// TIA Portal V17 export
// export: Created 2025-03-07T09:16:45.6631924Z, ExportSetting WithDefaults, DisplayName Totally Integrated Automation Portal, DisplayVersion V17 Update 8, DisplayName TIA Portal Openness, DisplayVersion V17 Update 8, DisplayName TIA Portal Version Control Interface, DisplayVersion V17, DisplayName SINAMICS Startdrive Advanced, DisplayVersion V17 SP2, DisplayName SINAMICS Startdrive G110M, G120, G120C, G120D, G120P, G115D, DisplayVersion V17 SP2, DisplayName SINAMICS Startdrive G130, G150, S120, S150, SINAMICS MV, S210, DisplayVersion V17 SP2, DisplayName STEP 7 Professional, DisplayVersion V17 Update 8, DisplayName SINUMERIK ONE STEP 7 Toolbox, DisplayVersion V17 Update 12, DisplayName SINUMERIK 840D sl STEP 7 Toolbox, DisplayVersion V17 Update 12, DisplayName STEP 7 Safety, DisplayVersion V17 Update 6, DisplayName WinCC Advanced, DisplayVersion V17 Update 8
FUNCTION "FC2800_UNIT_01_FIXTURE_4" : Void   // FC2800, LAD
TITLE = FIXTURE 1
{ S7_Optimized_Access := 'FALSE' }
AUTHOR : ETXETAR
VERSION : 1.0
// stored: AutoNumber false, IsIECCheckEnabled false, SetENOAutomatically false, UDAEnableTagReadback false
   VAR CONSTANT
      FC_NUMBER : DInt := 2800;
   END_VAR
   VAR_TEMP   // added for the SCL form of the ladder/FBD networks
      _w1 : Bool;
      _w2 : Bool;
      _w3 : Bool;
      _w4 : Bool;
      _w5 : Bool;
   END_VAR
BEGIN

REGION Network 1: PART A PRESENT INPUT
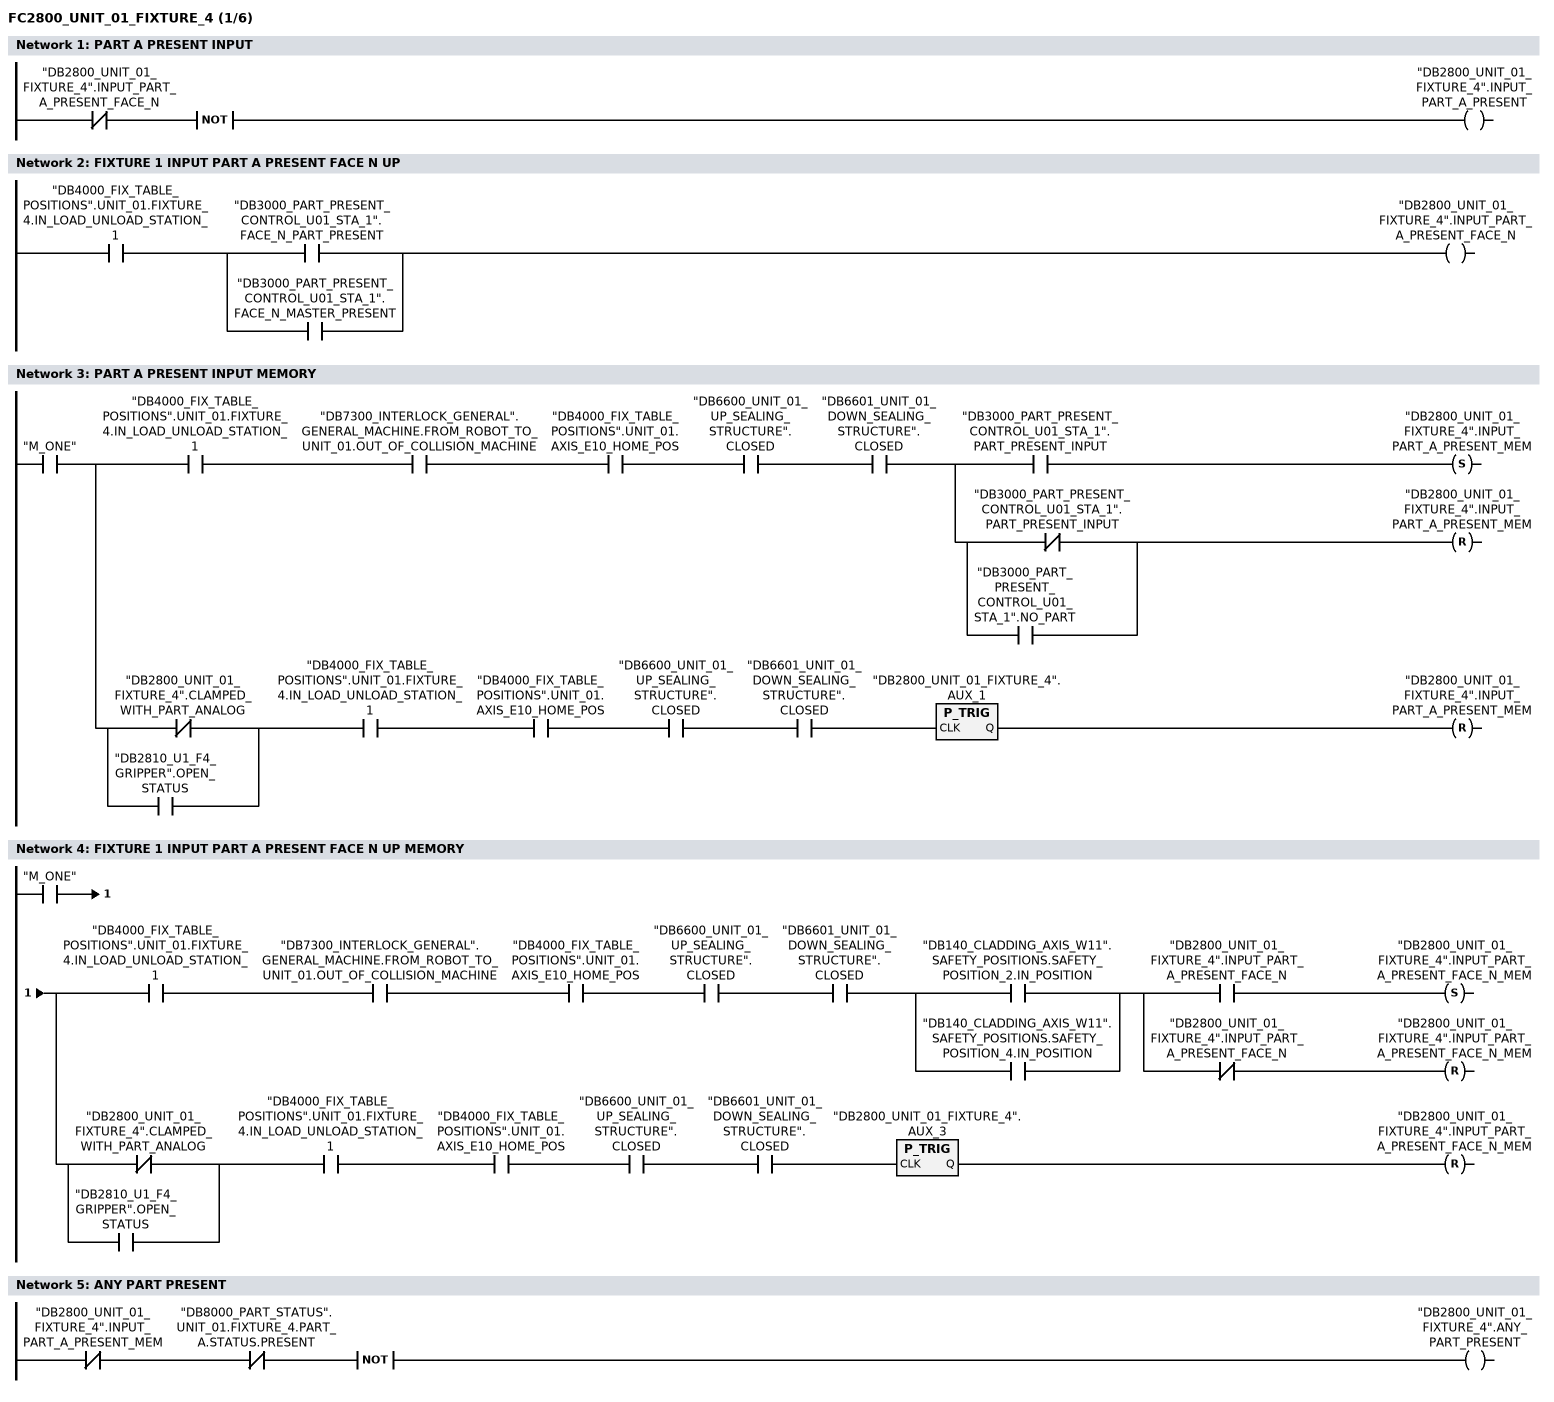
   RUNG wire#powerrail
      I_Contact( "DB2800_UNIT_01_FIXTURE_4".INPUT_PART_A_PRESENT_FACE_N )
      Not()
      Coil( "DB2800_UNIT_01_FIXTURE_4".INPUT_PART_A_PRESENT )
   END_RUNG
   // the same network as SCL:
   "DB2800_UNIT_01_FIXTURE_4".INPUT_PART_A_PRESENT := NOT (NOT "DB2800_UNIT_01_FIXTURE_4".INPUT_PART_A_PRESENT_FACE_N);
END_REGION

REGION Network 2: FIXTURE 1 INPUT PART A PRESENT FACE N UP
   RUNG wire#powerrail
      Contact( "DB4000_FIX_TABLE_POSITIONS".UNIT_01.FIXTURE_4.IN_LOAD_UNLOAD_STATION_1 )
      wire#w1
      Contact( "DB3000_PART_PRESENT_CONTROL_U01_STA_1".FACE_N_PART_PRESENT )
      wire#w2
      Coil( "DB2800_UNIT_01_FIXTURE_4".INPUT_PART_A_PRESENT_FACE_N )
   END_RUNG
   RUNG wire#w1
      Contact( "DB3000_PART_PRESENT_CONTROL_U01_STA_1".FACE_N_MASTER_PRESENT )
   END_RUNG wire#w2
   // the same network as SCL:
   "DB2800_UNIT_01_FIXTURE_4".INPUT_PART_A_PRESENT_FACE_N := "DB4000_FIX_TABLE_POSITIONS".UNIT_01.FIXTURE_4.IN_LOAD_UNLOAD_STATION_1 AND ("DB3000_PART_PRESENT_CONTROL_U01_STA_1".FACE_N_PART_PRESENT OR "DB3000_PART_PRESENT_CONTROL_U01_STA_1".FACE_N_MASTER_PRESENT);
END_REGION

REGION Network 3: PART A PRESENT INPUT MEMORY
   RUNG wire#powerrail
      Contact( "M_ONE" )
      wire#w1
      Contact( "DB4000_FIX_TABLE_POSITIONS".UNIT_01.FIXTURE_4.IN_LOAD_UNLOAD_STATION_1 )
      Contact( "DB7300_INTERLOCK_GENERAL".GENERAL_MACHINE.FROM_ROBOT_TO_UNIT_01.OUT_OF_COLLISION_MACHINE )
      Contact( "DB4000_FIX_TABLE_POSITIONS".UNIT_01.AXIS_E10_HOME_POS )
      Contact( "DB6600_UNIT_01_UP_SEALING_STRUCTURE".CLOSED )
      Contact( "DB6601_UNIT_01_DOWN_SEALING_STRUCTURE".CLOSED )
      wire#w2
      Contact( "DB3000_PART_PRESENT_CONTROL_U01_STA_1".PART_PRESENT_INPUT )
      S_Coil( "DB2800_UNIT_01_FIXTURE_4".INPUT_PART_A_PRESENT_MEM )
   END_RUNG
   RUNG wire#w2
      I_Contact( "DB3000_PART_PRESENT_CONTROL_U01_STA_1".PART_PRESENT_INPUT )
      wire#w3
      R_Coil( "DB2800_UNIT_01_FIXTURE_4".INPUT_PART_A_PRESENT_MEM )
   END_RUNG
   RUNG wire#w2
      Contact( "DB3000_PART_PRESENT_CONTROL_U01_STA_1".NO_PART )
   END_RUNG wire#w3
   RUNG wire#w1
      I_Contact( "DB2800_UNIT_01_FIXTURE_4".CLAMPED_WITH_PART_ANALOG )
      wire#w4
      Contact( "DB4000_FIX_TABLE_POSITIONS".UNIT_01.FIXTURE_4.IN_LOAD_UNLOAD_STATION_1 )
      Contact( "DB4000_FIX_TABLE_POSITIONS".UNIT_01.AXIS_E10_HOME_POS )
      Contact( "DB6600_UNIT_01_UP_SEALING_STRUCTURE".CLOSED )
      Contact( "DB6601_UNIT_01_DOWN_SEALING_STRUCTURE".CLOSED )
      P_Trig( "DB2800_UNIT_01_FIXTURE_4".AUX_1 )
      R_Coil( "DB2800_UNIT_01_FIXTURE_4".INPUT_PART_A_PRESENT_MEM )
   END_RUNG
   RUNG wire#w1
      Contact( "DB2810_U1_F4_GRIPPER".OPEN_STATUS )
   END_RUNG wire#w4
   // the same network as SCL:
   #_w1 := "M_ONE" AND "DB4000_FIX_TABLE_POSITIONS".UNIT_01.FIXTURE_4.IN_LOAD_UNLOAD_STATION_1 AND "DB7300_INTERLOCK_GENERAL".GENERAL_MACHINE.FROM_ROBOT_TO_UNIT_01.OUT_OF_COLLISION_MACHINE AND "DB4000_FIX_TABLE_POSITIONS".UNIT_01.AXIS_E10_HOME_POS AND "DB6600_UNIT_01_UP_SEALING_STRUCTURE".CLOSED AND "DB6601_UNIT_01_DOWN_SEALING_STRUCTURE".CLOSED;
   IF #_w1 AND "DB3000_PART_PRESENT_CONTROL_U01_STA_1".PART_PRESENT_INPUT THEN
       "DB2800_UNIT_01_FIXTURE_4".INPUT_PART_A_PRESENT_MEM := TRUE;
   END_IF;
   IF #_w1 AND (NOT "DB3000_PART_PRESENT_CONTROL_U01_STA_1".PART_PRESENT_INPUT OR "DB3000_PART_PRESENT_CONTROL_U01_STA_1".NO_PART) THEN
       "DB2800_UNIT_01_FIXTURE_4".INPUT_PART_A_PRESENT_MEM := FALSE;
   END_IF;
   #_w2 := "M_ONE" AND (NOT "DB2800_UNIT_01_FIXTURE_4".CLAMPED_WITH_PART_ANALOG OR "DB2810_U1_F4_GRIPPER".OPEN_STATUS) AND "DB4000_FIX_TABLE_POSITIONS".UNIT_01.FIXTURE_4.IN_LOAD_UNLOAD_STATION_1 AND "DB4000_FIX_TABLE_POSITIONS".UNIT_01.AXIS_E10_HOME_POS AND "DB6600_UNIT_01_UP_SEALING_STRUCTURE".CLOSED AND "DB6601_UNIT_01_DOWN_SEALING_STRUCTURE".CLOSED;
   #_w3 := #_w2 AND NOT "DB2800_UNIT_01_FIXTURE_4".AUX_1;   // rising edge
   "DB2800_UNIT_01_FIXTURE_4".AUX_1 := #_w2;
   IF #_w3 THEN "DB2800_UNIT_01_FIXTURE_4".INPUT_PART_A_PRESENT_MEM := FALSE; END_IF;
END_REGION

REGION Network 4: FIXTURE 1 INPUT PART A PRESENT FACE N UP MEMORY
   RUNG wire#powerrail
      Contact( "M_ONE" )
      wire#w1
      Contact( "DB4000_FIX_TABLE_POSITIONS".UNIT_01.FIXTURE_4.IN_LOAD_UNLOAD_STATION_1 )
      Contact( "DB7300_INTERLOCK_GENERAL".GENERAL_MACHINE.FROM_ROBOT_TO_UNIT_01.OUT_OF_COLLISION_MACHINE )
      Contact( "DB4000_FIX_TABLE_POSITIONS".UNIT_01.AXIS_E10_HOME_POS )
      Contact( "DB6600_UNIT_01_UP_SEALING_STRUCTURE".CLOSED )
      Contact( "DB6601_UNIT_01_DOWN_SEALING_STRUCTURE".CLOSED )
      wire#w2
      Contact( "DB140_CLADDING_AXIS_W11".SAFETY_POSITIONS.SAFETY_POSITION_2.IN_POSITION )
      wire#w3
      Contact( "DB2800_UNIT_01_FIXTURE_4".INPUT_PART_A_PRESENT_FACE_N )
      S_Coil( "DB2800_UNIT_01_FIXTURE_4".INPUT_PART_A_PRESENT_FACE_N_MEM )
   END_RUNG
   RUNG wire#w2
      Contact( "DB140_CLADDING_AXIS_W11".SAFETY_POSITIONS.SAFETY_POSITION_4.IN_POSITION )
   END_RUNG wire#w3
   RUNG wire#w3
      I_Contact( "DB2800_UNIT_01_FIXTURE_4".INPUT_PART_A_PRESENT_FACE_N )
      R_Coil( "DB2800_UNIT_01_FIXTURE_4".INPUT_PART_A_PRESENT_FACE_N_MEM )
   END_RUNG
   RUNG wire#w1
      I_Contact( "DB2800_UNIT_01_FIXTURE_4".CLAMPED_WITH_PART_ANALOG )
      wire#w4
      Contact( "DB4000_FIX_TABLE_POSITIONS".UNIT_01.FIXTURE_4.IN_LOAD_UNLOAD_STATION_1 )
      Contact( "DB4000_FIX_TABLE_POSITIONS".UNIT_01.AXIS_E10_HOME_POS )
      Contact( "DB6600_UNIT_01_UP_SEALING_STRUCTURE".CLOSED )
      Contact( "DB6601_UNIT_01_DOWN_SEALING_STRUCTURE".CLOSED )
      P_Trig( "DB2800_UNIT_01_FIXTURE_4".AUX_3 )
      R_Coil( "DB2800_UNIT_01_FIXTURE_4".INPUT_PART_A_PRESENT_FACE_N_MEM )
   END_RUNG
   RUNG wire#w1
      Contact( "DB2810_U1_F4_GRIPPER".OPEN_STATUS )
   END_RUNG wire#w4
   // the same network as SCL:
   #_w1 := "M_ONE" AND "DB4000_FIX_TABLE_POSITIONS".UNIT_01.FIXTURE_4.IN_LOAD_UNLOAD_STATION_1 AND "DB7300_INTERLOCK_GENERAL".GENERAL_MACHINE.FROM_ROBOT_TO_UNIT_01.OUT_OF_COLLISION_MACHINE AND "DB4000_FIX_TABLE_POSITIONS".UNIT_01.AXIS_E10_HOME_POS AND "DB6600_UNIT_01_UP_SEALING_STRUCTURE".CLOSED AND "DB6601_UNIT_01_DOWN_SEALING_STRUCTURE".CLOSED AND ("DB140_CLADDING_AXIS_W11".SAFETY_POSITIONS.SAFETY_POSITION_2.IN_POSITION OR "DB140_CLADDING_AXIS_W11".SAFETY_POSITIONS.SAFETY_POSITION_4.IN_POSITION);
   IF #_w1 AND "DB2800_UNIT_01_FIXTURE_4".INPUT_PART_A_PRESENT_FACE_N THEN
       "DB2800_UNIT_01_FIXTURE_4".INPUT_PART_A_PRESENT_FACE_N_MEM := TRUE;
   END_IF;
   IF #_w1 AND NOT "DB2800_UNIT_01_FIXTURE_4".INPUT_PART_A_PRESENT_FACE_N THEN
       "DB2800_UNIT_01_FIXTURE_4".INPUT_PART_A_PRESENT_FACE_N_MEM := FALSE;
   END_IF;
   #_w2 := "M_ONE" AND (NOT "DB2800_UNIT_01_FIXTURE_4".CLAMPED_WITH_PART_ANALOG OR "DB2810_U1_F4_GRIPPER".OPEN_STATUS) AND "DB4000_FIX_TABLE_POSITIONS".UNIT_01.FIXTURE_4.IN_LOAD_UNLOAD_STATION_1 AND "DB4000_FIX_TABLE_POSITIONS".UNIT_01.AXIS_E10_HOME_POS AND "DB6600_UNIT_01_UP_SEALING_STRUCTURE".CLOSED AND "DB6601_UNIT_01_DOWN_SEALING_STRUCTURE".CLOSED;
   #_w3 := #_w2 AND NOT "DB2800_UNIT_01_FIXTURE_4".AUX_3;   // rising edge
   "DB2800_UNIT_01_FIXTURE_4".AUX_3 := #_w2;
   IF #_w3 THEN "DB2800_UNIT_01_FIXTURE_4".INPUT_PART_A_PRESENT_FACE_N_MEM := FALSE; END_IF;
END_REGION

REGION Network 5: ANY PART PRESENT
   RUNG wire#powerrail
      I_Contact( "DB2800_UNIT_01_FIXTURE_4".INPUT_PART_A_PRESENT_MEM )
      I_Contact( "DB8000_PART_STATUS".UNIT_01.FIXTURE_4.PART_A.STATUS.PRESENT )
      Not()
      Coil( "DB2800_UNIT_01_FIXTURE_4".ANY_PART_PRESENT )
   END_RUNG
   // the same network as SCL:
   "DB2800_UNIT_01_FIXTURE_4".ANY_PART_PRESENT := NOT (NOT "DB2800_UNIT_01_FIXTURE_4".INPUT_PART_A_PRESENT_MEM AND NOT "DB8000_PART_STATUS".UNIT_01.FIXTURE_4.PART_A.STATUS.PRESENT);
END_REGION

REGION Network 6: CLAMPED WITH PART A
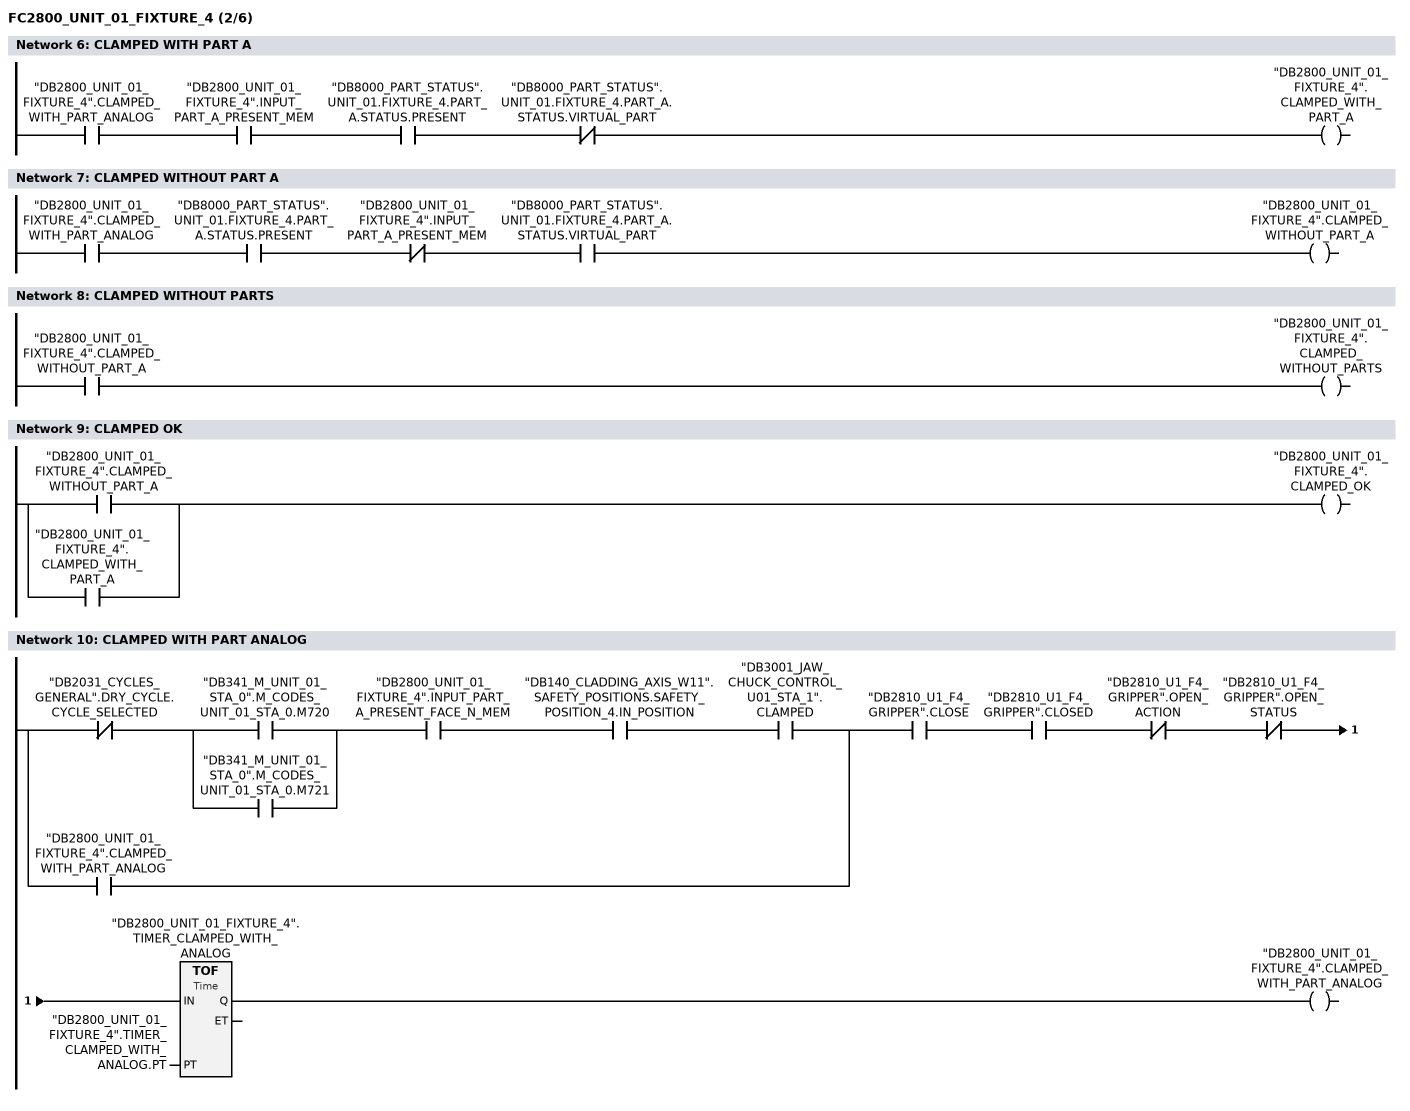
   RUNG wire#powerrail
      Contact( "DB2800_UNIT_01_FIXTURE_4".CLAMPED_WITH_PART_ANALOG )
      Contact( "DB2800_UNIT_01_FIXTURE_4".INPUT_PART_A_PRESENT_MEM )
      Contact( "DB8000_PART_STATUS".UNIT_01.FIXTURE_4.PART_A.STATUS.PRESENT )
      I_Contact( "DB8000_PART_STATUS".UNIT_01.FIXTURE_4.PART_A.STATUS.VIRTUAL_PART )
      Coil( "DB2800_UNIT_01_FIXTURE_4".CLAMPED_WITH_PART_A )
   END_RUNG
   // the same network as SCL:
   "DB2800_UNIT_01_FIXTURE_4".CLAMPED_WITH_PART_A := "DB2800_UNIT_01_FIXTURE_4".CLAMPED_WITH_PART_ANALOG AND "DB2800_UNIT_01_FIXTURE_4".INPUT_PART_A_PRESENT_MEM AND "DB8000_PART_STATUS".UNIT_01.FIXTURE_4.PART_A.STATUS.PRESENT AND NOT "DB8000_PART_STATUS".UNIT_01.FIXTURE_4.PART_A.STATUS.VIRTUAL_PART;
END_REGION

REGION Network 7: CLAMPED WITHOUT PART A
   RUNG wire#powerrail
      Contact( "DB2800_UNIT_01_FIXTURE_4".CLAMPED_WITH_PART_ANALOG )
      Contact( "DB8000_PART_STATUS".UNIT_01.FIXTURE_4.PART_A.STATUS.PRESENT )
      I_Contact( "DB2800_UNIT_01_FIXTURE_4".INPUT_PART_A_PRESENT_MEM )
      Contact( "DB8000_PART_STATUS".UNIT_01.FIXTURE_4.PART_A.STATUS.VIRTUAL_PART )
      Coil( "DB2800_UNIT_01_FIXTURE_4".CLAMPED_WITHOUT_PART_A )
   END_RUNG
   // the same network as SCL:
   "DB2800_UNIT_01_FIXTURE_4".CLAMPED_WITHOUT_PART_A := "DB2800_UNIT_01_FIXTURE_4".CLAMPED_WITH_PART_ANALOG AND "DB8000_PART_STATUS".UNIT_01.FIXTURE_4.PART_A.STATUS.PRESENT AND NOT "DB2800_UNIT_01_FIXTURE_4".INPUT_PART_A_PRESENT_MEM AND "DB8000_PART_STATUS".UNIT_01.FIXTURE_4.PART_A.STATUS.VIRTUAL_PART;
END_REGION

REGION Network 8: CLAMPED WITHOUT PARTS
   RUNG wire#powerrail
      Contact( "DB2800_UNIT_01_FIXTURE_4".CLAMPED_WITHOUT_PART_A )
      Coil( "DB2800_UNIT_01_FIXTURE_4".CLAMPED_WITHOUT_PARTS )
   END_RUNG
   // the same network as SCL:
   "DB2800_UNIT_01_FIXTURE_4".CLAMPED_WITHOUT_PARTS := "DB2800_UNIT_01_FIXTURE_4".CLAMPED_WITHOUT_PART_A;
END_REGION

REGION Network 9: CLAMPED OK
   RUNG wire#powerrail
      Contact( "DB2800_UNIT_01_FIXTURE_4".CLAMPED_WITHOUT_PART_A )
      wire#w1
      Coil( "DB2800_UNIT_01_FIXTURE_4".CLAMPED_OK )
   END_RUNG
   RUNG wire#powerrail
      Contact( "DB2800_UNIT_01_FIXTURE_4".CLAMPED_WITH_PART_A )
   END_RUNG wire#w1
   // the same network as SCL:
   "DB2800_UNIT_01_FIXTURE_4".CLAMPED_OK := "DB2800_UNIT_01_FIXTURE_4".CLAMPED_WITHOUT_PART_A OR "DB2800_UNIT_01_FIXTURE_4".CLAMPED_WITH_PART_A;
END_REGION

REGION Network 10: CLAMPED WITH PART ANALOG
   RUNG wire#powerrail
      I_Contact( "DB2031_CYCLES_GENERAL".DRY_CYCLE.CYCLE_SELECTED )
      wire#w1
      Contact( "DB341_M_UNIT_01_STA_0".M_CODES_UNIT_01_STA_0.M720 )
      wire#w2
      Contact( "DB2800_UNIT_01_FIXTURE_4".INPUT_PART_A_PRESENT_FACE_N_MEM )
      Contact( "DB140_CLADDING_AXIS_W11".SAFETY_POSITIONS.SAFETY_POSITION_4.IN_POSITION )
      Contact( "DB3001_JAW_CHUCK_CONTROL_U01_STA_1".CLAMPED )
      wire#w3
      Contact( "DB2810_U1_F4_GRIPPER".CLOSE )
      Contact( "DB2810_U1_F4_GRIPPER".CLOSED )
      I_Contact( "DB2810_U1_F4_GRIPPER".OPEN_ACTION )
      I_Contact( "DB2810_U1_F4_GRIPPER".OPEN_STATUS )
      { S7_Templates := "time_type := Time" } "DB2800_UNIT_01_FIXTURE_4".TIMER_CLAMPED_WITH_ANALOG.TOF(pt := "DB2800_UNIT_01_FIXTURE_4".TIMER_CLAMPED_WITH_ANALOG.PT, et =>)
      Coil( "DB2800_UNIT_01_FIXTURE_4".CLAMPED_WITH_PART_ANALOG )
   END_RUNG
   RUNG wire#w1
      Contact( "DB341_M_UNIT_01_STA_0".M_CODES_UNIT_01_STA_0.M721 )
   END_RUNG wire#w2
   RUNG wire#powerrail
      Contact( "DB2800_UNIT_01_FIXTURE_4".CLAMPED_WITH_PART_ANALOG )
   END_RUNG wire#w3
   // the same network as SCL:
   "DB2800_UNIT_01_FIXTURE_4".TIMER_CLAMPED_WITH_ANALOG.TOF(IN := ((NOT "DB2031_CYCLES_GENERAL".DRY_CYCLE.CYCLE_SELECTED AND ("DB341_M_UNIT_01_STA_0".M_CODES_UNIT_01_STA_0.M720 OR "DB341_M_UNIT_01_STA_0".M_CODES_UNIT_01_STA_0.M721) AND "DB2800_UNIT_01_FIXTURE_4".INPUT_PART_A_PRESENT_FACE_N_MEM AND "DB140_CLADDING_AXIS_W11".SAFETY_POSITIONS.SAFETY_POSITION_4.IN_POSITION AND "DB3001_JAW_CHUCK_CONTROL_U01_STA_1".CLAMPED) OR "DB2800_UNIT_01_FIXTURE_4".CLAMPED_WITH_PART_ANALOG) AND "DB2810_U1_F4_GRIPPER".CLOSE AND "DB2810_U1_F4_GRIPPER".CLOSED AND NOT "DB2810_U1_F4_GRIPPER".OPEN_ACTION AND NOT "DB2810_U1_F4_GRIPPER".OPEN_STATUS,
                           PT := "DB2800_UNIT_01_FIXTURE_4".TIMER_CLAMPED_WITH_ANALOG.PT);
   "DB2800_UNIT_01_FIXTURE_4".CLAMPED_WITH_PART_ANALOG := "DB2800_UNIT_01_FIXTURE_4".TIMER_CLAMPED_WITH_ANALOG.Q;
END_REGION

REGION Network 11: CLAMPED WITHOUT PART ANALOG
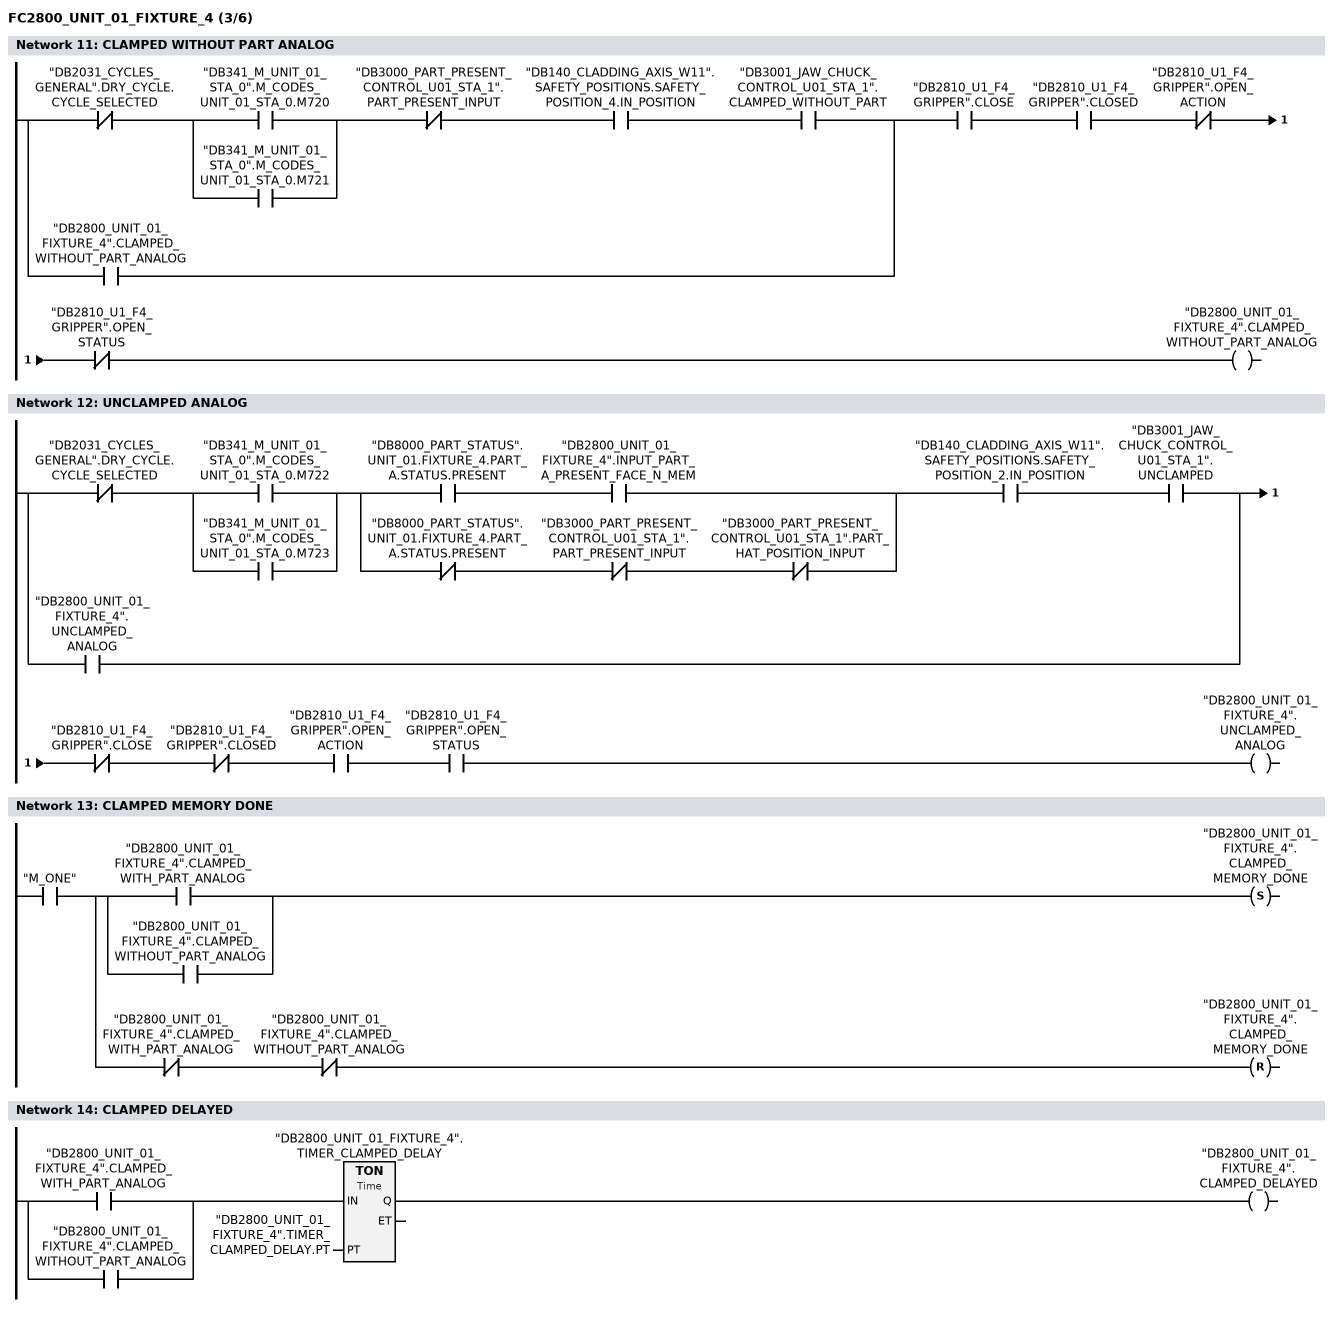
   RUNG wire#powerrail
      I_Contact( "DB2031_CYCLES_GENERAL".DRY_CYCLE.CYCLE_SELECTED )
      wire#w1
      Contact( "DB341_M_UNIT_01_STA_0".M_CODES_UNIT_01_STA_0.M720 )
      wire#w2
      I_Contact( "DB3000_PART_PRESENT_CONTROL_U01_STA_1".PART_PRESENT_INPUT )
      Contact( "DB140_CLADDING_AXIS_W11".SAFETY_POSITIONS.SAFETY_POSITION_4.IN_POSITION )
      Contact( "DB3001_JAW_CHUCK_CONTROL_U01_STA_1".CLAMPED_WITHOUT_PART )
      wire#w3
      Contact( "DB2810_U1_F4_GRIPPER".CLOSE )
      Contact( "DB2810_U1_F4_GRIPPER".CLOSED )
      I_Contact( "DB2810_U1_F4_GRIPPER".OPEN_ACTION )
      I_Contact( "DB2810_U1_F4_GRIPPER".OPEN_STATUS )
      Coil( "DB2800_UNIT_01_FIXTURE_4".CLAMPED_WITHOUT_PART_ANALOG )
   END_RUNG
   RUNG wire#w1
      Contact( "DB341_M_UNIT_01_STA_0".M_CODES_UNIT_01_STA_0.M721 )
   END_RUNG wire#w2
   RUNG wire#powerrail
      Contact( "DB2800_UNIT_01_FIXTURE_4".CLAMPED_WITHOUT_PART_ANALOG )
   END_RUNG wire#w3
   // the same network as SCL:
   "DB2800_UNIT_01_FIXTURE_4".CLAMPED_WITHOUT_PART_ANALOG := ((NOT "DB2031_CYCLES_GENERAL".DRY_CYCLE.CYCLE_SELECTED AND ("DB341_M_UNIT_01_STA_0".M_CODES_UNIT_01_STA_0.M720 OR "DB341_M_UNIT_01_STA_0".M_CODES_UNIT_01_STA_0.M721) AND NOT "DB3000_PART_PRESENT_CONTROL_U01_STA_1".PART_PRESENT_INPUT AND "DB140_CLADDING_AXIS_W11".SAFETY_POSITIONS.SAFETY_POSITION_4.IN_POSITION AND "DB3001_JAW_CHUCK_CONTROL_U01_STA_1".CLAMPED_WITHOUT_PART) OR "DB2800_UNIT_01_FIXTURE_4".CLAMPED_WITHOUT_PART_ANALOG) AND "DB2810_U1_F4_GRIPPER".CLOSE AND "DB2810_U1_F4_GRIPPER".CLOSED AND NOT "DB2810_U1_F4_GRIPPER".OPEN_ACTION AND NOT "DB2810_U1_F4_GRIPPER".OPEN_STATUS;
END_REGION

REGION Network 12: UNCLAMPED ANALOG
   RUNG wire#powerrail
      I_Contact( "DB2031_CYCLES_GENERAL".DRY_CYCLE.CYCLE_SELECTED )
      wire#w1
      Contact( "DB341_M_UNIT_01_STA_0".M_CODES_UNIT_01_STA_0.M722 )
      wire#w2
      Contact( "DB8000_PART_STATUS".UNIT_01.FIXTURE_4.PART_A.STATUS.PRESENT )
      Contact( "DB2800_UNIT_01_FIXTURE_4".INPUT_PART_A_PRESENT_FACE_N_MEM )
      wire#w3
      Contact( "DB140_CLADDING_AXIS_W11".SAFETY_POSITIONS.SAFETY_POSITION_2.IN_POSITION )
      Contact( "DB3001_JAW_CHUCK_CONTROL_U01_STA_1".UNCLAMPED )
      wire#w4
      I_Contact( "DB2810_U1_F4_GRIPPER".CLOSE )
      I_Contact( "DB2810_U1_F4_GRIPPER".CLOSED )
      Contact( "DB2810_U1_F4_GRIPPER".OPEN_ACTION )
      Contact( "DB2810_U1_F4_GRIPPER".OPEN_STATUS )
      Coil( "DB2800_UNIT_01_FIXTURE_4".UNCLAMPED_ANALOG )
   END_RUNG
   RUNG wire#w1
      Contact( "DB341_M_UNIT_01_STA_0".M_CODES_UNIT_01_STA_0.M723 )
   END_RUNG wire#w2
   RUNG wire#w2
      I_Contact( "DB8000_PART_STATUS".UNIT_01.FIXTURE_4.PART_A.STATUS.PRESENT )
      I_Contact( "DB3000_PART_PRESENT_CONTROL_U01_STA_1".PART_PRESENT_INPUT )
      I_Contact( "DB3000_PART_PRESENT_CONTROL_U01_STA_1".PART_HAT_POSITION_INPUT )
   END_RUNG wire#w3
   RUNG wire#powerrail
      Contact( "DB2800_UNIT_01_FIXTURE_4".UNCLAMPED_ANALOG )
   END_RUNG wire#w4
   // the same network as SCL:
   "DB2800_UNIT_01_FIXTURE_4".UNCLAMPED_ANALOG := ((NOT "DB2031_CYCLES_GENERAL".DRY_CYCLE.CYCLE_SELECTED AND ("DB341_M_UNIT_01_STA_0".M_CODES_UNIT_01_STA_0.M722 OR "DB341_M_UNIT_01_STA_0".M_CODES_UNIT_01_STA_0.M723) AND (("DB8000_PART_STATUS".UNIT_01.FIXTURE_4.PART_A.STATUS.PRESENT AND "DB2800_UNIT_01_FIXTURE_4".INPUT_PART_A_PRESENT_FACE_N_MEM) OR (NOT "DB8000_PART_STATUS".UNIT_01.FIXTURE_4.PART_A.STATUS.PRESENT AND NOT "DB3000_PART_PRESENT_CONTROL_U01_STA_1".PART_PRESENT_INPUT AND NOT "DB3000_PART_PRESENT_CONTROL_U01_STA_1".PART_HAT_POSITION_INPUT)) AND "DB140_CLADDING_AXIS_W11".SAFETY_POSITIONS.SAFETY_POSITION_2.IN_POSITION AND "DB3001_JAW_CHUCK_CONTROL_U01_STA_1".UNCLAMPED) OR "DB2800_UNIT_01_FIXTURE_4".UNCLAMPED_ANALOG) AND NOT "DB2810_U1_F4_GRIPPER".CLOSE AND NOT "DB2810_U1_F4_GRIPPER".CLOSED AND "DB2810_U1_F4_GRIPPER".OPEN_ACTION AND "DB2810_U1_F4_GRIPPER".OPEN_STATUS;
END_REGION

REGION Network 13: CLAMPED MEMORY DONE
   RUNG wire#powerrail
      Contact( "M_ONE" )
      wire#w1
      Contact( "DB2800_UNIT_01_FIXTURE_4".CLAMPED_WITH_PART_ANALOG )
      wire#w2
      S_Coil( "DB2800_UNIT_01_FIXTURE_4".CLAMPED_MEMORY_DONE )
   END_RUNG
   RUNG wire#w1
      Contact( "DB2800_UNIT_01_FIXTURE_4".CLAMPED_WITHOUT_PART_ANALOG )
   END_RUNG wire#w2
   RUNG wire#w1
      I_Contact( "DB2800_UNIT_01_FIXTURE_4".CLAMPED_WITH_PART_ANALOG )
      I_Contact( "DB2800_UNIT_01_FIXTURE_4".CLAMPED_WITHOUT_PART_ANALOG )
      R_Coil( "DB2800_UNIT_01_FIXTURE_4".CLAMPED_MEMORY_DONE )
   END_RUNG
   // the same network as SCL:
   IF "M_ONE" AND ("DB2800_UNIT_01_FIXTURE_4".CLAMPED_WITH_PART_ANALOG OR "DB2800_UNIT_01_FIXTURE_4".CLAMPED_WITHOUT_PART_ANALOG) THEN
       "DB2800_UNIT_01_FIXTURE_4".CLAMPED_MEMORY_DONE := TRUE;
   END_IF;
   IF "M_ONE" AND NOT "DB2800_UNIT_01_FIXTURE_4".CLAMPED_WITH_PART_ANALOG AND NOT "DB2800_UNIT_01_FIXTURE_4".CLAMPED_WITHOUT_PART_ANALOG THEN
       "DB2800_UNIT_01_FIXTURE_4".CLAMPED_MEMORY_DONE := FALSE;
   END_IF;
END_REGION

REGION Network 14: CLAMPED DELAYED
   RUNG wire#powerrail
      Contact( "DB2800_UNIT_01_FIXTURE_4".CLAMPED_WITH_PART_ANALOG )
      wire#w1
      { S7_Templates := "time_type := Time" } "DB2800_UNIT_01_FIXTURE_4".TIMER_CLAMPED_DELAY.TON(pt := "DB2800_UNIT_01_FIXTURE_4".TIMER_CLAMPED_DELAY.PT, et =>)
      Coil( "DB2800_UNIT_01_FIXTURE_4".CLAMPED_DELAYED )
   END_RUNG
   RUNG wire#powerrail
      Contact( "DB2800_UNIT_01_FIXTURE_4".CLAMPED_WITHOUT_PART_ANALOG )
   END_RUNG wire#w1
   // the same network as SCL:
   "DB2800_UNIT_01_FIXTURE_4".TIMER_CLAMPED_DELAY.TON(IN := "DB2800_UNIT_01_FIXTURE_4".CLAMPED_WITH_PART_ANALOG OR "DB2800_UNIT_01_FIXTURE_4".CLAMPED_WITHOUT_PART_ANALOG,
                           PT := "DB2800_UNIT_01_FIXTURE_4".TIMER_CLAMPED_DELAY.PT);
   "DB2800_UNIT_01_FIXTURE_4".CLAMPED_DELAYED := "DB2800_UNIT_01_FIXTURE_4".TIMER_CLAMPED_DELAY.Q;
END_REGION

REGION Network 15: ALL CNC PLC VARIABLES ZERO
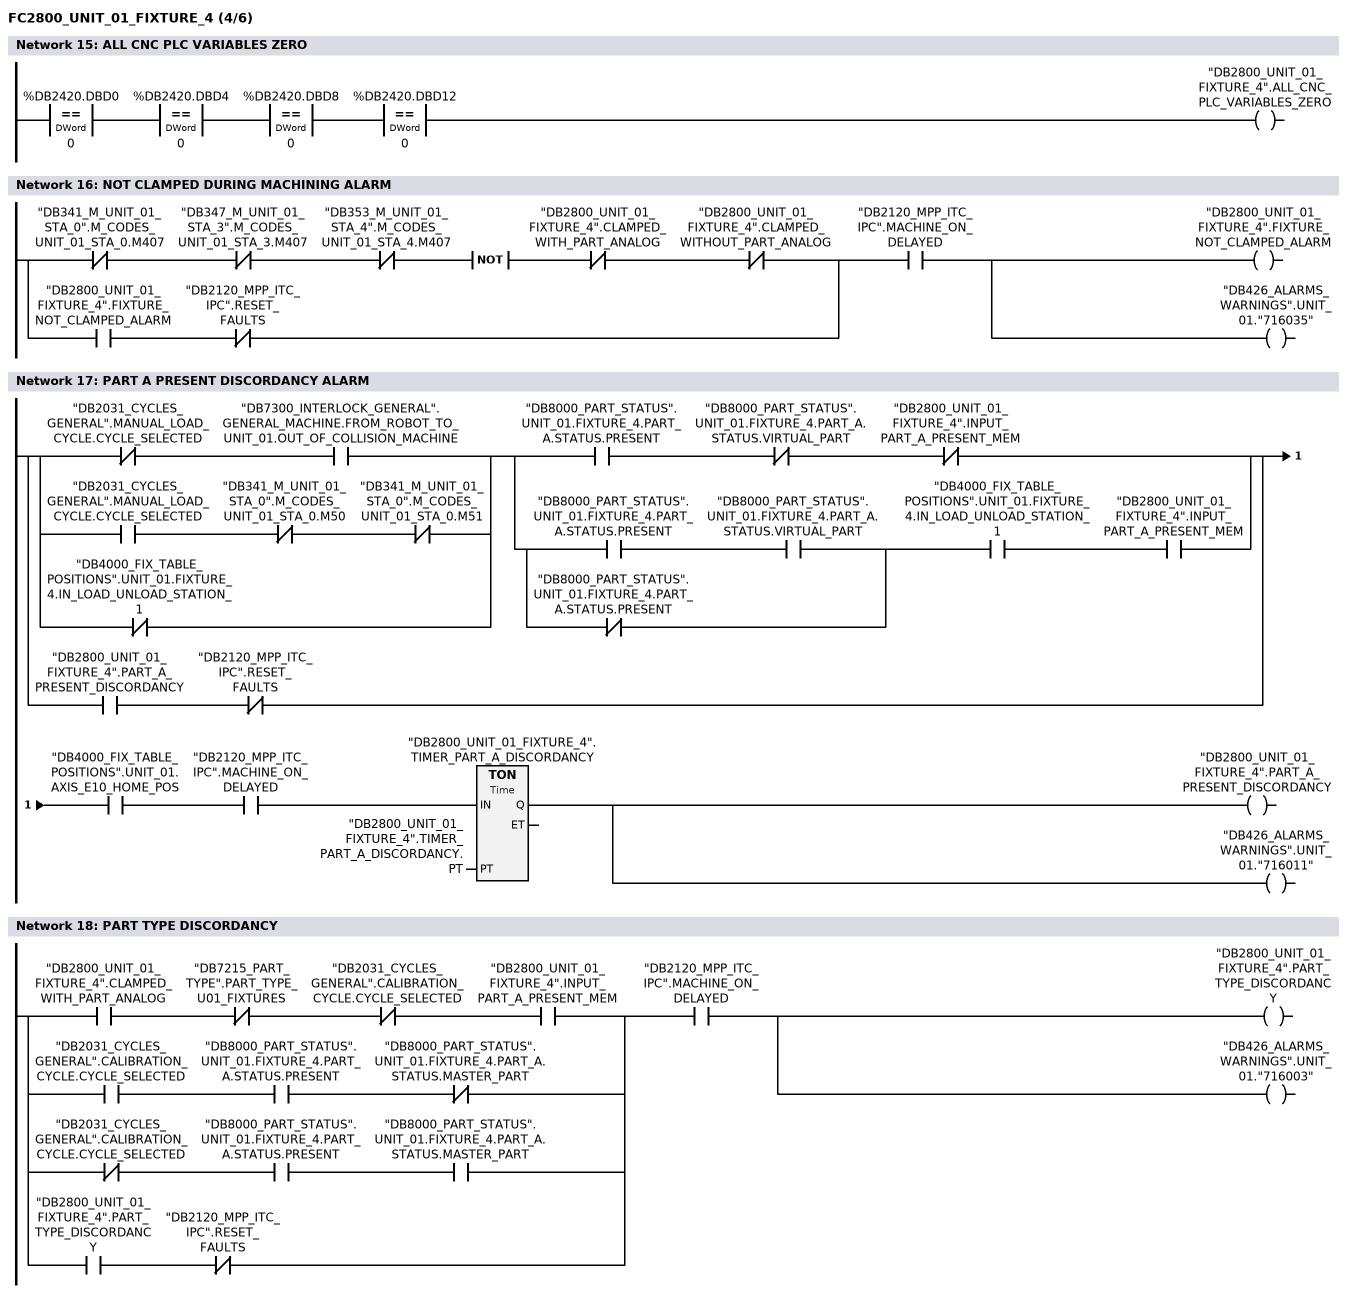
   RUNG wire#powerrail
      { S7_Templates := "SrcType := DWord" } EQ_Contact(in1 := %DB2420.DBD0, in2 := 0)
      { S7_Templates := "SrcType := DWord" } EQ_Contact(in1 := %DB2420.DBD4, in2 := 0)
      { S7_Templates := "SrcType := DWord" } EQ_Contact(in1 := %DB2420.DBD8, in2 := 0)
      { S7_Templates := "SrcType := DWord" } EQ_Contact(in1 := %DB2420.DBD12, in2 := 0)
      Coil( "DB2800_UNIT_01_FIXTURE_4".ALL_CNC_PLC_VARIABLES_ZERO )
   END_RUNG
   // the same network as SCL:
   "DB2800_UNIT_01_FIXTURE_4".ALL_CNC_PLC_VARIABLES_ZERO := (%DB2420.DBD0 = 0) AND (%DB2420.DBD4 = 0) AND (%DB2420.DBD8 = 0) AND (%DB2420.DBD12 = 0);
END_REGION

REGION Network 16: NOT CLAMPED DURING MACHINING ALARM
   RUNG wire#powerrail
      I_Contact( "DB341_M_UNIT_01_STA_0".M_CODES_UNIT_01_STA_0.M407 )
      I_Contact( "DB347_M_UNIT_01_STA_3".M_CODES_UNIT_01_STA_3.M407 )
      I_Contact( "DB353_M_UNIT_01_STA_4".M_CODES_UNIT_01_STA_4.M407 )
      Not()
      I_Contact( "DB2800_UNIT_01_FIXTURE_4".CLAMPED_WITH_PART_ANALOG )
      I_Contact( "DB2800_UNIT_01_FIXTURE_4".CLAMPED_WITHOUT_PART_ANALOG )
      wire#w1
      Contact( "DB2120_MPP_ITC_IPC".MACHINE_ON_DELAYED )
      wire#w2
      Coil( "DB2800_UNIT_01_FIXTURE_4".FIXTURE_NOT_CLAMPED_ALARM )
   END_RUNG
   RUNG wire#powerrail
      Contact( "DB2800_UNIT_01_FIXTURE_4".FIXTURE_NOT_CLAMPED_ALARM )
      I_Contact( "DB2120_MPP_ITC_IPC".RESET_FAULTS )
   END_RUNG wire#w1
   RUNG wire#w2
      Coil( "DB426_ALARMS_WARNINGS".UNIT_01."716035" )
   END_RUNG
   // the same network as SCL:
   "DB2800_UNIT_01_FIXTURE_4".FIXTURE_NOT_CLAMPED_ALARM := ((NOT (NOT "DB341_M_UNIT_01_STA_0".M_CODES_UNIT_01_STA_0.M407 AND NOT "DB347_M_UNIT_01_STA_3".M_CODES_UNIT_01_STA_3.M407 AND NOT "DB353_M_UNIT_01_STA_4".M_CODES_UNIT_01_STA_4.M407) AND NOT "DB2800_UNIT_01_FIXTURE_4".CLAMPED_WITH_PART_ANALOG AND NOT "DB2800_UNIT_01_FIXTURE_4".CLAMPED_WITHOUT_PART_ANALOG) OR ("DB2800_UNIT_01_FIXTURE_4".FIXTURE_NOT_CLAMPED_ALARM AND NOT "DB2120_MPP_ITC_IPC".RESET_FAULTS)) AND "DB2120_MPP_ITC_IPC".MACHINE_ON_DELAYED;
   "DB426_ALARMS_WARNINGS".UNIT_01."716035" := "DB2800_UNIT_01_FIXTURE_4".FIXTURE_NOT_CLAMPED_ALARM;
END_REGION

REGION Network 17: PART A PRESENT DISCORDANCY ALARM
   RUNG wire#powerrail
      I_Contact( "DB2031_CYCLES_GENERAL".MANUAL_LOAD_CYCLE.CYCLE_SELECTED )
      Contact( "DB7300_INTERLOCK_GENERAL".GENERAL_MACHINE.FROM_ROBOT_TO_UNIT_01.OUT_OF_COLLISION_MACHINE )
      wire#w1
      Contact( "DB8000_PART_STATUS".UNIT_01.FIXTURE_4.PART_A.STATUS.PRESENT )
      I_Contact( "DB8000_PART_STATUS".UNIT_01.FIXTURE_4.PART_A.STATUS.VIRTUAL_PART )
      I_Contact( "DB2800_UNIT_01_FIXTURE_4".INPUT_PART_A_PRESENT_MEM )
      wire#w2
      Contact( "DB4000_FIX_TABLE_POSITIONS".UNIT_01.AXIS_E10_HOME_POS )
      Contact( "DB2120_MPP_ITC_IPC".MACHINE_ON_DELAYED )
      { S7_Templates := "time_type := Time" } "DB2800_UNIT_01_FIXTURE_4".TIMER_PART_A_DISCORDANCY.TON(pt := "DB2800_UNIT_01_FIXTURE_4".TIMER_PART_A_DISCORDANCY.PT, et =>)
      wire#w4
      Coil( "DB2800_UNIT_01_FIXTURE_4".PART_A_PRESENT_DISCORDANCY )
   END_RUNG
   RUNG wire#powerrail
      Contact( "DB2031_CYCLES_GENERAL".MANUAL_LOAD_CYCLE.CYCLE_SELECTED )
      I_Contact( "DB341_M_UNIT_01_STA_0".M_CODES_UNIT_01_STA_0.M50 )
      I_Contact( "DB341_M_UNIT_01_STA_0".M_CODES_UNIT_01_STA_0.M51 )
   END_RUNG wire#w1
   RUNG wire#powerrail
      I_Contact( "DB4000_FIX_TABLE_POSITIONS".UNIT_01.FIXTURE_4.IN_LOAD_UNLOAD_STATION_1 )
   END_RUNG wire#w1
   RUNG wire#w1
      Contact( "DB8000_PART_STATUS".UNIT_01.FIXTURE_4.PART_A.STATUS.PRESENT )
      Contact( "DB8000_PART_STATUS".UNIT_01.FIXTURE_4.PART_A.STATUS.VIRTUAL_PART )
      wire#w3
      Contact( "DB4000_FIX_TABLE_POSITIONS".UNIT_01.FIXTURE_4.IN_LOAD_UNLOAD_STATION_1 )
      Contact( "DB2800_UNIT_01_FIXTURE_4".INPUT_PART_A_PRESENT_MEM )
   END_RUNG wire#w2
   RUNG wire#w1
      I_Contact( "DB8000_PART_STATUS".UNIT_01.FIXTURE_4.PART_A.STATUS.PRESENT )
   END_RUNG wire#w3
   RUNG wire#powerrail
      Contact( "DB2800_UNIT_01_FIXTURE_4".PART_A_PRESENT_DISCORDANCY )
      I_Contact( "DB2120_MPP_ITC_IPC".RESET_FAULTS )
   END_RUNG wire#w2
   RUNG wire#w4
      Coil( "DB426_ALARMS_WARNINGS".UNIT_01."716011" )
   END_RUNG
   // the same network as SCL:
   "DB2800_UNIT_01_FIXTURE_4".TIMER_PART_A_DISCORDANCY.TON(IN := ((((NOT "DB2031_CYCLES_GENERAL".MANUAL_LOAD_CYCLE.CYCLE_SELECTED AND "DB7300_INTERLOCK_GENERAL".GENERAL_MACHINE.FROM_ROBOT_TO_UNIT_01.OUT_OF_COLLISION_MACHINE) OR ("DB2031_CYCLES_GENERAL".MANUAL_LOAD_CYCLE.CYCLE_SELECTED AND NOT "DB341_M_UNIT_01_STA_0".M_CODES_UNIT_01_STA_0.M50 AND NOT "DB341_M_UNIT_01_STA_0".M_CODES_UNIT_01_STA_0.M51) OR NOT "DB4000_FIX_TABLE_POSITIONS".UNIT_01.FIXTURE_4.IN_LOAD_UNLOAD_STATION_1) AND (("DB8000_PART_STATUS".UNIT_01.FIXTURE_4.PART_A.STATUS.PRESENT AND NOT "DB8000_PART_STATUS".UNIT_01.FIXTURE_4.PART_A.STATUS.VIRTUAL_PART AND NOT "DB2800_UNIT_01_FIXTURE_4".INPUT_PART_A_PRESENT_MEM) OR ((("DB8000_PART_STATUS".UNIT_01.FIXTURE_4.PART_A.STATUS.PRESENT AND "DB8000_PART_STATUS".UNIT_01.FIXTURE_4.PART_A.STATUS.VIRTUAL_PART) OR NOT "DB8000_PART_STATUS".UNIT_01.FIXTURE_4.PART_A.STATUS.PRESENT) AND "DB4000_FIX_TABLE_POSITIONS".UNIT_01.FIXTURE_4.IN_LOAD_UNLOAD_STATION_1 AND "DB2800_UNIT_01_FIXTURE_4".INPUT_PART_A_PRESENT_MEM))) OR ("DB2800_UNIT_01_FIXTURE_4".PART_A_PRESENT_DISCORDANCY AND NOT "DB2120_MPP_ITC_IPC".RESET_FAULTS)) AND "DB4000_FIX_TABLE_POSITIONS".UNIT_01.AXIS_E10_HOME_POS AND "DB2120_MPP_ITC_IPC".MACHINE_ON_DELAYED,
                           PT := "DB2800_UNIT_01_FIXTURE_4".TIMER_PART_A_DISCORDANCY.PT);
   "DB2800_UNIT_01_FIXTURE_4".PART_A_PRESENT_DISCORDANCY := "DB2800_UNIT_01_FIXTURE_4".TIMER_PART_A_DISCORDANCY.Q;
   "DB426_ALARMS_WARNINGS".UNIT_01."716011" := "DB2800_UNIT_01_FIXTURE_4".TIMER_PART_A_DISCORDANCY.Q;
END_REGION

REGION Network 18: PART TYPE DISCORDANCY
   RUNG wire#powerrail
      Contact( "DB2800_UNIT_01_FIXTURE_4".CLAMPED_WITH_PART_ANALOG )
      I_Contact( "DB7215_PART_TYPE".PART_TYPE_U01_FIXTURES )
      I_Contact( "DB2031_CYCLES_GENERAL".CALIBRATION_CYCLE.CYCLE_SELECTED )
      Contact( "DB2800_UNIT_01_FIXTURE_4".INPUT_PART_A_PRESENT_MEM )
      wire#w1
      Contact( "DB2120_MPP_ITC_IPC".MACHINE_ON_DELAYED )
      wire#w2
      Coil( "DB2800_UNIT_01_FIXTURE_4".PART_TYPE_DISCORDANCY )
   END_RUNG
   RUNG wire#powerrail
      Contact( "DB2031_CYCLES_GENERAL".CALIBRATION_CYCLE.CYCLE_SELECTED )
      Contact( "DB8000_PART_STATUS".UNIT_01.FIXTURE_4.PART_A.STATUS.PRESENT )
      I_Contact( "DB8000_PART_STATUS".UNIT_01.FIXTURE_4.PART_A.STATUS.MASTER_PART )
   END_RUNG wire#w1
   RUNG wire#powerrail
      I_Contact( "DB2031_CYCLES_GENERAL".CALIBRATION_CYCLE.CYCLE_SELECTED )
      Contact( "DB8000_PART_STATUS".UNIT_01.FIXTURE_4.PART_A.STATUS.PRESENT )
      Contact( "DB8000_PART_STATUS".UNIT_01.FIXTURE_4.PART_A.STATUS.MASTER_PART )
   END_RUNG wire#w1
   RUNG wire#powerrail
      Contact( "DB2800_UNIT_01_FIXTURE_4".PART_TYPE_DISCORDANCY )
      I_Contact( "DB2120_MPP_ITC_IPC".RESET_FAULTS )
   END_RUNG wire#w1
   RUNG wire#w2
      Coil( "DB426_ALARMS_WARNINGS".UNIT_01."716003" )
   END_RUNG
   // the same network as SCL:
   "DB2800_UNIT_01_FIXTURE_4".PART_TYPE_DISCORDANCY := (("DB2800_UNIT_01_FIXTURE_4".CLAMPED_WITH_PART_ANALOG AND NOT "DB7215_PART_TYPE".PART_TYPE_U01_FIXTURES AND NOT "DB2031_CYCLES_GENERAL".CALIBRATION_CYCLE.CYCLE_SELECTED AND "DB2800_UNIT_01_FIXTURE_4".INPUT_PART_A_PRESENT_MEM) OR ("DB2031_CYCLES_GENERAL".CALIBRATION_CYCLE.CYCLE_SELECTED AND "DB8000_PART_STATUS".UNIT_01.FIXTURE_4.PART_A.STATUS.PRESENT AND NOT "DB8000_PART_STATUS".UNIT_01.FIXTURE_4.PART_A.STATUS.MASTER_PART) OR (NOT "DB2031_CYCLES_GENERAL".CALIBRATION_CYCLE.CYCLE_SELECTED AND "DB8000_PART_STATUS".UNIT_01.FIXTURE_4.PART_A.STATUS.PRESENT AND "DB8000_PART_STATUS".UNIT_01.FIXTURE_4.PART_A.STATUS.MASTER_PART) OR ("DB2800_UNIT_01_FIXTURE_4".PART_TYPE_DISCORDANCY AND NOT "DB2120_MPP_ITC_IPC".RESET_FAULTS)) AND "DB2120_MPP_ITC_IPC".MACHINE_ON_DELAYED;
   "DB426_ALARMS_WARNINGS".UNIT_01."716003" := "DB2800_UNIT_01_FIXTURE_4".PART_TYPE_DISCORDANCY;
END_REGION

REGION Network 19: PART A ORIENTATED DISCORDANCY
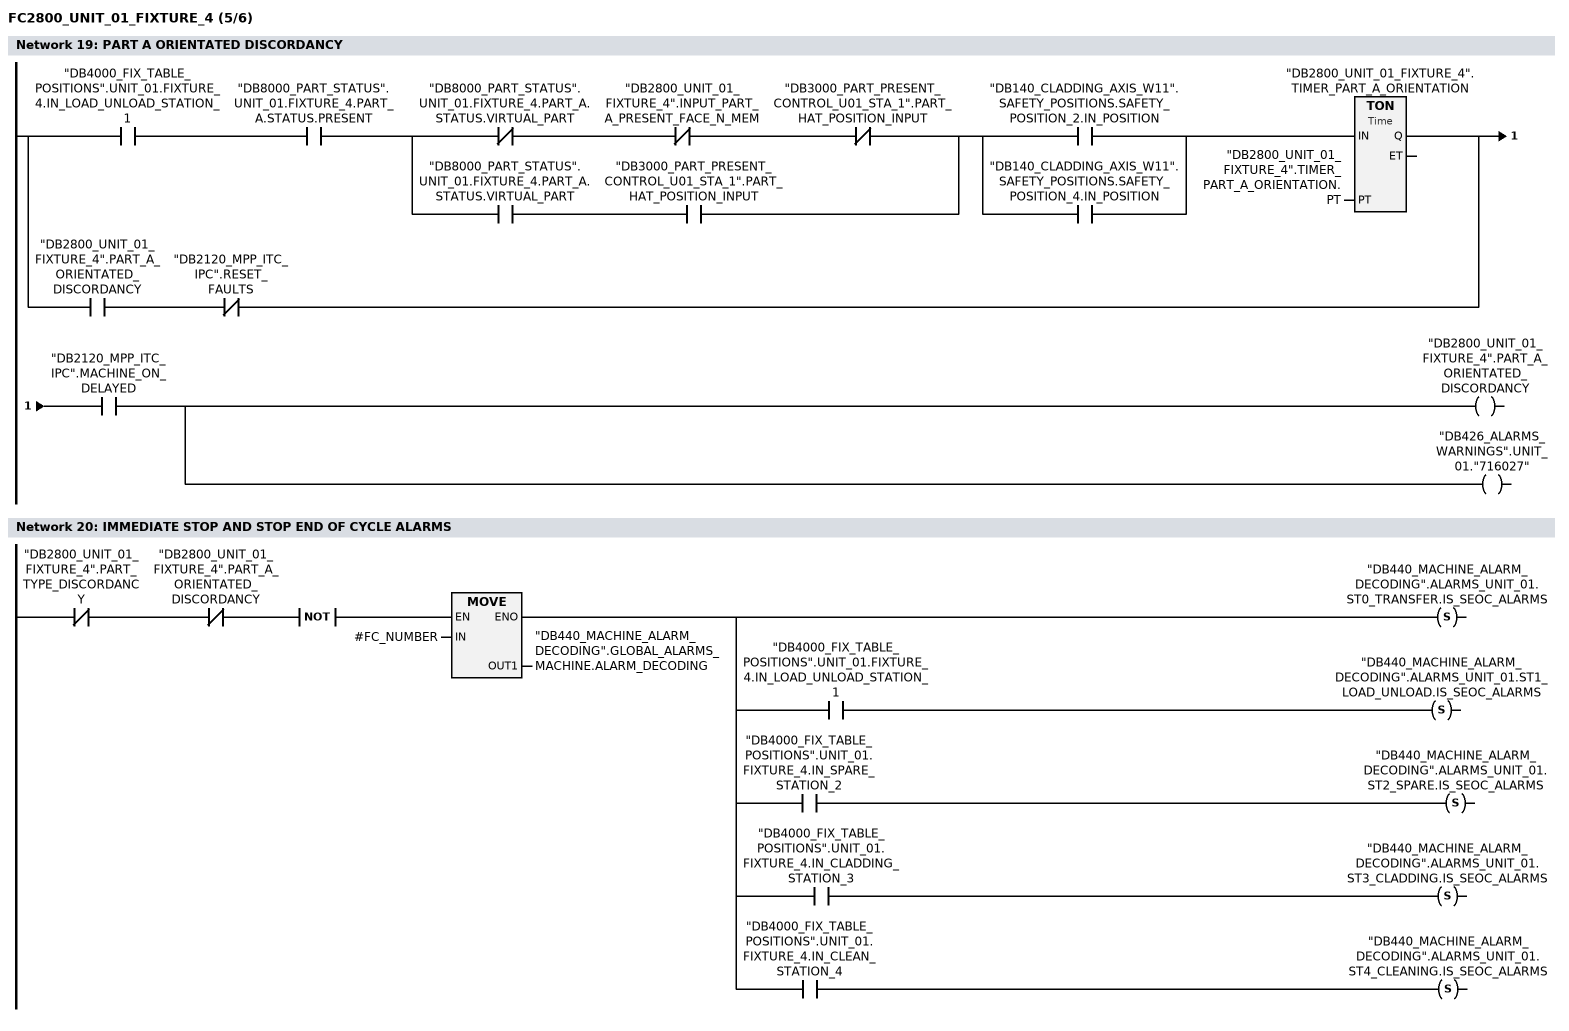
   RUNG wire#powerrail
      Contact( "DB4000_FIX_TABLE_POSITIONS".UNIT_01.FIXTURE_4.IN_LOAD_UNLOAD_STATION_1 )
      Contact( "DB8000_PART_STATUS".UNIT_01.FIXTURE_4.PART_A.STATUS.PRESENT )
      wire#w1
      I_Contact( "DB8000_PART_STATUS".UNIT_01.FIXTURE_4.PART_A.STATUS.VIRTUAL_PART )
      I_Contact( "DB2800_UNIT_01_FIXTURE_4".INPUT_PART_A_PRESENT_FACE_N_MEM )
      I_Contact( "DB3000_PART_PRESENT_CONTROL_U01_STA_1".PART_HAT_POSITION_INPUT )
      wire#w2
      Contact( "DB140_CLADDING_AXIS_W11".SAFETY_POSITIONS.SAFETY_POSITION_2.IN_POSITION )
      wire#w3
      { S7_Templates := "time_type := Time" } "DB2800_UNIT_01_FIXTURE_4".TIMER_PART_A_ORIENTATION.TON(pt := "DB2800_UNIT_01_FIXTURE_4".TIMER_PART_A_ORIENTATION.PT, et =>)
      wire#w4
      Contact( "DB2120_MPP_ITC_IPC".MACHINE_ON_DELAYED )
      wire#w5
      Coil( "DB2800_UNIT_01_FIXTURE_4".PART_A_ORIENTATED_DISCORDANCY )
   END_RUNG
   RUNG wire#w1
      Contact( "DB8000_PART_STATUS".UNIT_01.FIXTURE_4.PART_A.STATUS.VIRTUAL_PART )
      Contact( "DB3000_PART_PRESENT_CONTROL_U01_STA_1".PART_HAT_POSITION_INPUT )
   END_RUNG wire#w2
   RUNG wire#w2
      Contact( "DB140_CLADDING_AXIS_W11".SAFETY_POSITIONS.SAFETY_POSITION_4.IN_POSITION )
   END_RUNG wire#w3
   RUNG wire#powerrail
      Contact( "DB2800_UNIT_01_FIXTURE_4".PART_A_ORIENTATED_DISCORDANCY )
      I_Contact( "DB2120_MPP_ITC_IPC".RESET_FAULTS )
   END_RUNG wire#w4
   RUNG wire#w5
      Coil( "DB426_ALARMS_WARNINGS".UNIT_01."716027" )
   END_RUNG
   // the same network as SCL:
   "DB2800_UNIT_01_FIXTURE_4".TIMER_PART_A_ORIENTATION.TON(IN := "DB4000_FIX_TABLE_POSITIONS".UNIT_01.FIXTURE_4.IN_LOAD_UNLOAD_STATION_1 AND "DB8000_PART_STATUS".UNIT_01.FIXTURE_4.PART_A.STATUS.PRESENT AND ((NOT "DB8000_PART_STATUS".UNIT_01.FIXTURE_4.PART_A.STATUS.VIRTUAL_PART AND NOT "DB2800_UNIT_01_FIXTURE_4".INPUT_PART_A_PRESENT_FACE_N_MEM AND NOT "DB3000_PART_PRESENT_CONTROL_U01_STA_1".PART_HAT_POSITION_INPUT) OR ("DB8000_PART_STATUS".UNIT_01.FIXTURE_4.PART_A.STATUS.VIRTUAL_PART AND "DB3000_PART_PRESENT_CONTROL_U01_STA_1".PART_HAT_POSITION_INPUT)) AND ("DB140_CLADDING_AXIS_W11".SAFETY_POSITIONS.SAFETY_POSITION_2.IN_POSITION OR "DB140_CLADDING_AXIS_W11".SAFETY_POSITIONS.SAFETY_POSITION_4.IN_POSITION),
                           PT := "DB2800_UNIT_01_FIXTURE_4".TIMER_PART_A_ORIENTATION.PT);
   "DB2800_UNIT_01_FIXTURE_4".PART_A_ORIENTATED_DISCORDANCY := ("DB2800_UNIT_01_FIXTURE_4".TIMER_PART_A_ORIENTATION.Q OR ("DB2800_UNIT_01_FIXTURE_4".PART_A_ORIENTATED_DISCORDANCY AND NOT "DB2120_MPP_ITC_IPC".RESET_FAULTS)) AND "DB2120_MPP_ITC_IPC".MACHINE_ON_DELAYED;
   "DB426_ALARMS_WARNINGS".UNIT_01."716027" := "DB2800_UNIT_01_FIXTURE_4".PART_A_ORIENTATED_DISCORDANCY;
END_REGION

REGION Network 20: IMMEDIATE STOP AND STOP END OF CYCLE ALARMS
   RUNG wire#powerrail
      I_Contact( "DB2800_UNIT_01_FIXTURE_4".PART_TYPE_DISCORDANCY )
      I_Contact( "DB2800_UNIT_01_FIXTURE_4".PART_A_ORIENTATED_DISCORDANCY )
      Not()
      Move(in := #FC_NUMBER, out1 => "DB440_MACHINE_ALARM_DECODING".GLOBAL_ALARMS_MACHINE.ALARM_DECODING)
      wire#w1
      S_Coil( "DB440_MACHINE_ALARM_DECODING".ALARMS_UNIT_01.ST0_TRANSFER.IS_SEOC_ALARMS )
   END_RUNG
   RUNG wire#w1
      Contact( "DB4000_FIX_TABLE_POSITIONS".UNIT_01.FIXTURE_4.IN_LOAD_UNLOAD_STATION_1 )
      S_Coil( "DB440_MACHINE_ALARM_DECODING".ALARMS_UNIT_01.ST1_LOAD_UNLOAD.IS_SEOC_ALARMS )
   END_RUNG
   RUNG wire#w1
      Contact( "DB4000_FIX_TABLE_POSITIONS".UNIT_01.FIXTURE_4.IN_SPARE_STATION_2 )
      S_Coil( "DB440_MACHINE_ALARM_DECODING".ALARMS_UNIT_01.ST2_SPARE.IS_SEOC_ALARMS )
   END_RUNG
   RUNG wire#w1
      Contact( "DB4000_FIX_TABLE_POSITIONS".UNIT_01.FIXTURE_4.IN_CLADDING_STATION_3 )
      S_Coil( "DB440_MACHINE_ALARM_DECODING".ALARMS_UNIT_01.ST3_CLADDING.IS_SEOC_ALARMS )
   END_RUNG
   RUNG wire#w1
      Contact( "DB4000_FIX_TABLE_POSITIONS".UNIT_01.FIXTURE_4.IN_CLEAN_STATION_4 )
      S_Coil( "DB440_MACHINE_ALARM_DECODING".ALARMS_UNIT_01.ST4_CLEANING.IS_SEOC_ALARMS )
   END_RUNG
   // the same network as SCL:
   #_w1 := NOT (NOT "DB2800_UNIT_01_FIXTURE_4".PART_TYPE_DISCORDANCY AND NOT "DB2800_UNIT_01_FIXTURE_4".PART_A_ORIENTATED_DISCORDANCY);
   IF #_w1 THEN
       "DB440_MACHINE_ALARM_DECODING".GLOBAL_ALARMS_MACHINE.ALARM_DECODING := #FC_NUMBER;
       "DB440_MACHINE_ALARM_DECODING".ALARMS_UNIT_01.ST0_TRANSFER.IS_SEOC_ALARMS := TRUE;
   END_IF;
   IF #_w1 AND "DB4000_FIX_TABLE_POSITIONS".UNIT_01.FIXTURE_4.IN_LOAD_UNLOAD_STATION_1 THEN
       "DB440_MACHINE_ALARM_DECODING".ALARMS_UNIT_01.ST1_LOAD_UNLOAD.IS_SEOC_ALARMS := TRUE;
   END_IF;
   IF #_w1 AND "DB4000_FIX_TABLE_POSITIONS".UNIT_01.FIXTURE_4.IN_SPARE_STATION_2 THEN
       "DB440_MACHINE_ALARM_DECODING".ALARMS_UNIT_01.ST2_SPARE.IS_SEOC_ALARMS := TRUE;
   END_IF;
   IF #_w1 AND "DB4000_FIX_TABLE_POSITIONS".UNIT_01.FIXTURE_4.IN_CLADDING_STATION_3 THEN
       "DB440_MACHINE_ALARM_DECODING".ALARMS_UNIT_01.ST3_CLADDING.IS_SEOC_ALARMS := TRUE;
   END_IF;
   IF #_w1 AND "DB4000_FIX_TABLE_POSITIONS".UNIT_01.FIXTURE_4.IN_CLEAN_STATION_4 THEN
       "DB440_MACHINE_ALARM_DECODING".ALARMS_UNIT_01.ST4_CLEANING.IS_SEOC_ALARMS := TRUE;
   END_IF;
END_REGION

REGION Network 21: RETURN HOME POSITION AND STOP END OF CYCLE ALARMS
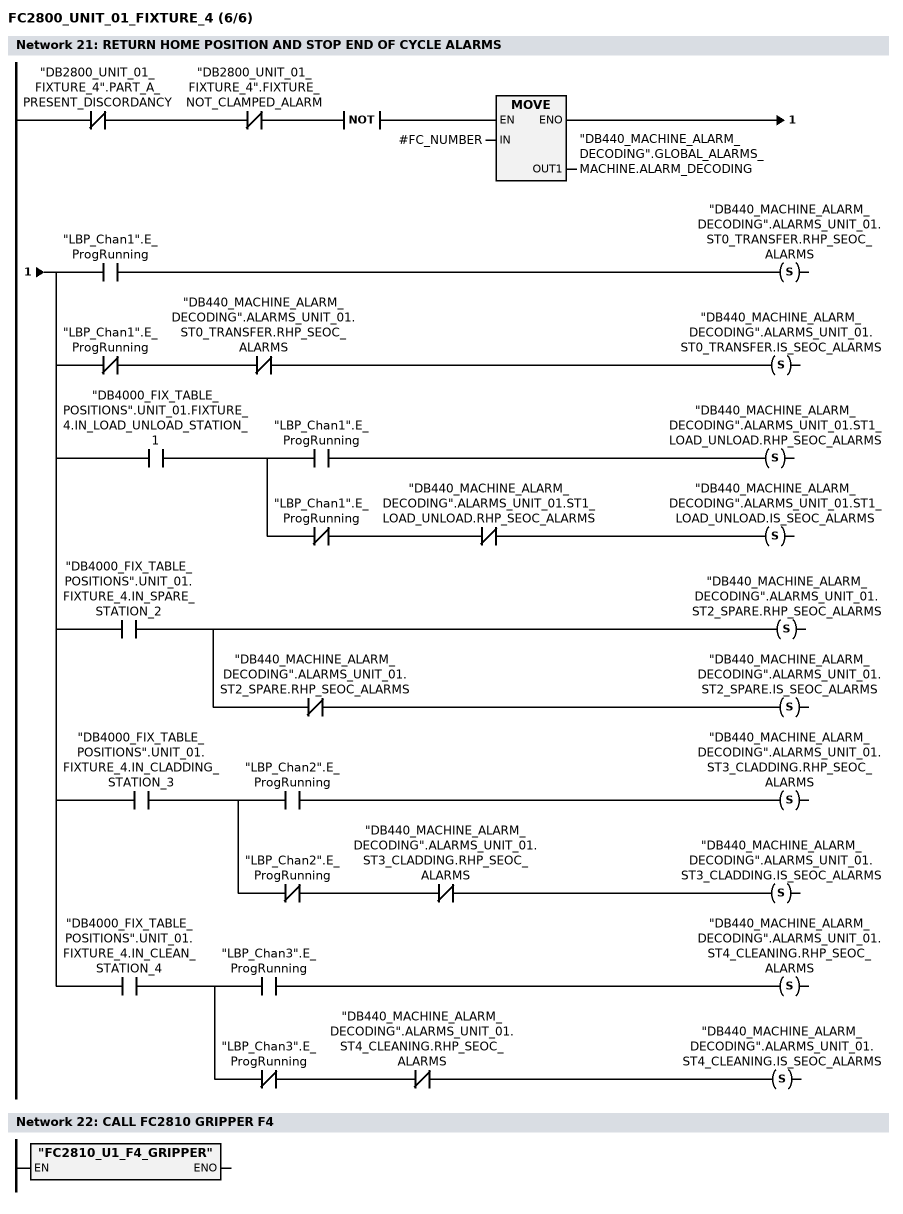
   RUNG wire#powerrail
      I_Contact( "DB2800_UNIT_01_FIXTURE_4".PART_A_PRESENT_DISCORDANCY )
      I_Contact( "DB2800_UNIT_01_FIXTURE_4".FIXTURE_NOT_CLAMPED_ALARM )
      Not()
      Move(in := #FC_NUMBER, out1 => "DB440_MACHINE_ALARM_DECODING".GLOBAL_ALARMS_MACHINE.ALARM_DECODING)
      wire#w1
      Contact( "LBP_Chan1".E_ProgRunning )
      S_Coil( "DB440_MACHINE_ALARM_DECODING".ALARMS_UNIT_01.ST0_TRANSFER.RHP_SEOC_ALARMS )
   END_RUNG
   RUNG wire#w1
      I_Contact( "LBP_Chan1".E_ProgRunning )
      I_Contact( "DB440_MACHINE_ALARM_DECODING".ALARMS_UNIT_01.ST0_TRANSFER.RHP_SEOC_ALARMS )
      S_Coil( "DB440_MACHINE_ALARM_DECODING".ALARMS_UNIT_01.ST0_TRANSFER.IS_SEOC_ALARMS )
   END_RUNG
   RUNG wire#w1
      Contact( "DB4000_FIX_TABLE_POSITIONS".UNIT_01.FIXTURE_4.IN_LOAD_UNLOAD_STATION_1 )
      wire#w2
      Contact( "LBP_Chan1".E_ProgRunning )
      S_Coil( "DB440_MACHINE_ALARM_DECODING".ALARMS_UNIT_01.ST1_LOAD_UNLOAD.RHP_SEOC_ALARMS )
   END_RUNG
   RUNG wire#w2
      I_Contact( "LBP_Chan1".E_ProgRunning )
      I_Contact( "DB440_MACHINE_ALARM_DECODING".ALARMS_UNIT_01.ST1_LOAD_UNLOAD.RHP_SEOC_ALARMS )
      S_Coil( "DB440_MACHINE_ALARM_DECODING".ALARMS_UNIT_01.ST1_LOAD_UNLOAD.IS_SEOC_ALARMS )
   END_RUNG
   RUNG wire#w1
      Contact( "DB4000_FIX_TABLE_POSITIONS".UNIT_01.FIXTURE_4.IN_SPARE_STATION_2 )
      wire#w3
      S_Coil( "DB440_MACHINE_ALARM_DECODING".ALARMS_UNIT_01.ST2_SPARE.RHP_SEOC_ALARMS )
   END_RUNG
   RUNG wire#w3
      I_Contact( "DB440_MACHINE_ALARM_DECODING".ALARMS_UNIT_01.ST2_SPARE.RHP_SEOC_ALARMS )
      S_Coil( "DB440_MACHINE_ALARM_DECODING".ALARMS_UNIT_01.ST2_SPARE.IS_SEOC_ALARMS )
   END_RUNG
   RUNG wire#w1
      Contact( "DB4000_FIX_TABLE_POSITIONS".UNIT_01.FIXTURE_4.IN_CLADDING_STATION_3 )
      wire#w4
      Contact( "LBP_Chan2".E_ProgRunning )
      S_Coil( "DB440_MACHINE_ALARM_DECODING".ALARMS_UNIT_01.ST3_CLADDING.RHP_SEOC_ALARMS )
   END_RUNG
   RUNG wire#w4
      I_Contact( "LBP_Chan2".E_ProgRunning )
      I_Contact( "DB440_MACHINE_ALARM_DECODING".ALARMS_UNIT_01.ST3_CLADDING.RHP_SEOC_ALARMS )
      S_Coil( "DB440_MACHINE_ALARM_DECODING".ALARMS_UNIT_01.ST3_CLADDING.IS_SEOC_ALARMS )
   END_RUNG
   RUNG wire#w1
      Contact( "DB4000_FIX_TABLE_POSITIONS".UNIT_01.FIXTURE_4.IN_CLEAN_STATION_4 )
      wire#w5
      Contact( "LBP_Chan3".E_ProgRunning )
      S_Coil( "DB440_MACHINE_ALARM_DECODING".ALARMS_UNIT_01.ST4_CLEANING.RHP_SEOC_ALARMS )
   END_RUNG
   RUNG wire#w5
      I_Contact( "LBP_Chan3".E_ProgRunning )
      I_Contact( "DB440_MACHINE_ALARM_DECODING".ALARMS_UNIT_01.ST4_CLEANING.RHP_SEOC_ALARMS )
      S_Coil( "DB440_MACHINE_ALARM_DECODING".ALARMS_UNIT_01.ST4_CLEANING.IS_SEOC_ALARMS )
   END_RUNG
   // the same network as SCL:
   #_w1 := NOT (NOT "DB2800_UNIT_01_FIXTURE_4".PART_A_PRESENT_DISCORDANCY AND NOT "DB2800_UNIT_01_FIXTURE_4".FIXTURE_NOT_CLAMPED_ALARM);
   IF #_w1 THEN "DB440_MACHINE_ALARM_DECODING".GLOBAL_ALARMS_MACHINE.ALARM_DECODING := #FC_NUMBER; END_IF;
   IF #_w1 AND "LBP_Chan1".E_ProgRunning THEN
       "DB440_MACHINE_ALARM_DECODING".ALARMS_UNIT_01.ST0_TRANSFER.RHP_SEOC_ALARMS := TRUE;
   END_IF;
   IF #_w1 AND NOT "LBP_Chan1".E_ProgRunning AND NOT "DB440_MACHINE_ALARM_DECODING".ALARMS_UNIT_01.ST0_TRANSFER.RHP_SEOC_ALARMS THEN
       "DB440_MACHINE_ALARM_DECODING".ALARMS_UNIT_01.ST0_TRANSFER.IS_SEOC_ALARMS := TRUE;
   END_IF;
   #_w2 := #_w1 AND "DB4000_FIX_TABLE_POSITIONS".UNIT_01.FIXTURE_4.IN_LOAD_UNLOAD_STATION_1;
   IF #_w2 AND "LBP_Chan1".E_ProgRunning THEN
       "DB440_MACHINE_ALARM_DECODING".ALARMS_UNIT_01.ST1_LOAD_UNLOAD.RHP_SEOC_ALARMS := TRUE;
   END_IF;
   IF #_w2 AND NOT "LBP_Chan1".E_ProgRunning AND NOT "DB440_MACHINE_ALARM_DECODING".ALARMS_UNIT_01.ST1_LOAD_UNLOAD.RHP_SEOC_ALARMS THEN
       "DB440_MACHINE_ALARM_DECODING".ALARMS_UNIT_01.ST1_LOAD_UNLOAD.IS_SEOC_ALARMS := TRUE;
   END_IF;
   #_w3 := #_w1 AND "DB4000_FIX_TABLE_POSITIONS".UNIT_01.FIXTURE_4.IN_SPARE_STATION_2;
   IF #_w3 THEN "DB440_MACHINE_ALARM_DECODING".ALARMS_UNIT_01.ST2_SPARE.RHP_SEOC_ALARMS := TRUE; END_IF;
   IF #_w3 AND NOT "DB440_MACHINE_ALARM_DECODING".ALARMS_UNIT_01.ST2_SPARE.RHP_SEOC_ALARMS THEN
       "DB440_MACHINE_ALARM_DECODING".ALARMS_UNIT_01.ST2_SPARE.IS_SEOC_ALARMS := TRUE;
   END_IF;
   #_w4 := #_w1 AND "DB4000_FIX_TABLE_POSITIONS".UNIT_01.FIXTURE_4.IN_CLADDING_STATION_3;
   IF #_w4 AND "LBP_Chan2".E_ProgRunning THEN
       "DB440_MACHINE_ALARM_DECODING".ALARMS_UNIT_01.ST3_CLADDING.RHP_SEOC_ALARMS := TRUE;
   END_IF;
   IF #_w4 AND NOT "LBP_Chan2".E_ProgRunning AND NOT "DB440_MACHINE_ALARM_DECODING".ALARMS_UNIT_01.ST3_CLADDING.RHP_SEOC_ALARMS THEN
       "DB440_MACHINE_ALARM_DECODING".ALARMS_UNIT_01.ST3_CLADDING.IS_SEOC_ALARMS := TRUE;
   END_IF;
   #_w5 := #_w1 AND "DB4000_FIX_TABLE_POSITIONS".UNIT_01.FIXTURE_4.IN_CLEAN_STATION_4;
   IF #_w5 AND "LBP_Chan3".E_ProgRunning THEN
       "DB440_MACHINE_ALARM_DECODING".ALARMS_UNIT_01.ST4_CLEANING.RHP_SEOC_ALARMS := TRUE;
   END_IF;
   IF #_w5 AND NOT "LBP_Chan3".E_ProgRunning AND NOT "DB440_MACHINE_ALARM_DECODING".ALARMS_UNIT_01.ST4_CLEANING.RHP_SEOC_ALARMS THEN
       "DB440_MACHINE_ALARM_DECODING".ALARMS_UNIT_01.ST4_CLEANING.IS_SEOC_ALARMS := TRUE;
   END_IF;
END_REGION

REGION Network 22: CALL FC2810 GRIPPER F4
   RUNG wire#powerrail
      "FC2810_U1_F4_GRIPPER"()
   END_RUNG
   // the same network as SCL:
   "FC2810_U1_F4_GRIPPER"();
END_REGION
END_FUNCTION
